(* PLC project Tc2_Utilities.FILETIME64_TO_TOD Demo, tc3-libraries-kb TwinCAT 3.1 *)
(* stored: creationDateTime 2026-05-10T12:00:00, modificationDateTime 2026-05-10T12:00:00 *)

PROGRAM P_Demo_FILETIME64_TO_TOD
  VAR
    rResult : TIME_OF_DAY;  (* FILETIME64_TO_TOD 的返回值 *)
    bRun : BOOL;  (* 触发一次调用 *)
    ftIn : T_FILETIME64;  (* 测试用本地变量 *)
  END_VAR

            // ============================================================
// Tc2_Utilities.FILETIME64_TO_TOD 演示程序（FUNCTION）
// ============================================================
// 验证步骤：
//   1. 引用 Tc2_Utilities（及类型所在依赖库 Tc2_System / Tc2_Standard）
//   2. 编译 + 登录
//   3. 强制 bRun := TRUE 一个周期
//   4. 观察 rResult 应为 TOD#12:34:56
// ============================================================

ftIn := DT_TO_FILETIME64(DT#2024-01-01-12:34:56);
IF bRun THEN
    rResult := FILETIME64_TO_TOD(ftIn);
    bRun := FALSE;
END_IF;

          
END_PROGRAM
